FUNCTION_BLOCK FB_AdsReader
VAR_INPUT
    sSymbol         : STRING;       // Symbol name to read e.g. 'GVL_Tank.nTankLevel'
    nPort           : UINT;         // Target PLC port e.g. 851
    tCycleTime      : TIME;         // How often to read e.g. T#500MS
    pDestAddr       : POINTER TO BYTE; // Pointer to local variable
    nDestSize       : UDINT;        // Size of local variable
END_VAR
VAR_OUTPUT
    bBusy           : BOOL;
    bError          : BOOL;
    nErrId          : UDINT;
    bNewValue       : BOOL;         // Pulses TRUE when fresh value arrives
END_VAR
VAR
	fbAdsHandle     : ADSRDWRTEX;
    fbAdsRead       : ADSREAD;
    fbCycleTimer    : TON;
    bTrigger        : BOOL;
   
END_VAR

END_FUNCTION_BLOCK

(* stored: Version 1.1.0.1, ProductVersion 3.1.4024.16
   POU Fb_AdsReader: Id {b4e92dd9-6112-4fac-b084-5b0a27fb5996}, SpecialFunc None *)
